Staubli VAL3: realTimeCtrl.dtx

public bool bActive = true
public bool bOverRun[3]
  [0] = true
  [1] = true
  [2] = true
public jointRx jJoint_RT_Start = {j1=50.2, j2=40, j3=75, j5=65}
public jointRx jNowJointPos
public jointRx jdJointPos
mdesc mMdesc_Init = {accel=25, vel=50, decel=25, tmax=500, rmax=99}
public mdesc mMdesc_RT = {accel=25, vel=50, decel=25, tmax=500, rmax=99, blend=off}
mdesc mNomSpeed
public num nDamp[6 6]
  [0,0] = 10
  [1,1] = 10
  [2,2] = 10
  [3,3] = 10
  [4,4] = 10
  [5,5] = 10
public num nFileID[6]
public num nForceTorque[6]
  [0] = -0.458435
  [1] = -0.0611247
  [2] = -0.0305157
  [3] = 0.00182448
  [4] = 0.00243784
public num nMass[6 6]
  [0,0] = 1
  [1,1] = 1
  [2,2] = 1
  [3,3] = 1
  [4,4] = 1
  [5,5] = 1
public num nNowCarteVel
public num nNowJointAccel[6]
public num nNowJointVel[6]
public num nNowPointAccel[6]
public num nNowPointVel[6]
public num nPort = 5001
public num nSensitivity[6]
  [0] = 32.72
  [1] = 32.72
  [2] = 32.77
  [3] = 1644.3
  [4] = 1640.8
  [5] = 1635
public num nSioTimeOut = 5
public num nStiffness[6 6]
  [0,0] = 25
  [1,1] = 25
  [2,2] = 25
  [3,3] = 25
  [4,4] = 25
  [5,5] = 25
public num nZeroPoint[6]
  [0] = 8211
  [1] = 8189
  [2] = 8176
  [3] = 8194
  [4] = 8176
  [5] = 8189
public num ndForceTorque[6]
public num ndJointAccel[6]
public num ndJointVel[6]
public num ndPointAccel[6]
public num ndPointVel[6]
public pointRx pNowPointPos = {fatherId=world[0]}
public pointRx pPointCommand = {fatherId=world[0]}
public pointRx pdPointPos = {fatherId=world[0]}
public sio sClient = {link=Socket\FTSensor}
tool tTool = {rz=180, fatherId=flange[0], ioLink=valve1}
